(* CODESYS project SNDLTN_HTTP.library
   Author: S. Verbeek
   Title: SNDLTN_HTTP
   Version: 1.2.200929
   Description: Library created to ease the use of the CoDeSys HTTP example.
   Company: Sandolution

Project tree, tasks and I/O mapping:
  libraries: CAA Net Base Services, * (CAA Technical Workgroup); CAA Behaviour Model, * (CAA Technical Workgroup); StringUtils, * (System); CAA Types, 3.0.0.1 (CAA Technical Workgroup)
  Constants/
    global variables HTTP_UTF8
    global variables HTTP_Properties
    global variables HTTP_Constants
  Enums/
    data type HTTP_eRequestType
    data type HTTP_eContentType
    data type HTTP_eError
    data type HTTP_eState_int
  Function Blocks/
    function block HTTP_Client [ST]: prvStart, StringToURL, prvCyclicAction, prvResetOutputs, CreateRequest, Close, prvAbort, ParseResult
  Functions/
    function HTTP_UTF8toUTF16_3S [ST]
    function HTTP_UTF16toUTF8_3S [ST]
    function HTTP_Concat_3S [ST]
    function HTTP_IsLegalUTF8_3S [ST]
  Structs/
    data type HTTP_scResponse
    data type HTTP_scURL_int
  Variables/
  program ChangeLog [ST]
*)

// Enums/HTTP_eRequestType
{attribute 'qualified_only'}
TYPE HTTP_eRequestType :
(
	GET := 0,
	POST, 		//(Requires pwsPostValue) 
	DELETE, 
	PUT,		//(Requires pwsPostValue) 
	HEAD
);
END_TYPE

// Enums/HTTP_eContentType
{attribute 'qualified_only'}
TYPE HTTP_eContentType :
(
	FORM := 0,		//HTTP FORM DATA
	JSON			//JSON/XML format
);
END_TYPE

// Enums/HTTP_eError
{attribute 'qualified_only'}
{attribute 'to_string'}
TYPE HTTP_eError :
(
	NoError 					:= 0, 		// No error
	
	//1000-1999 : HTTP ERRORS
	TCPInitError				:= 1001, 	// Unable to initialize the TCP socket
	TCPReadError				:= 1002, 	// Error while reading response
	TCPWriteError				:= 1003, 	// Error while sending the request
	MissingPostValue			:= 1004, 	// Current request type needs a post value
	ParsingError				:= 1005, 	// Error while parsing the response
	
	//NBS errors (ported from 6001-6099)
	NBS_TimeOut 				:= 1100,	//Time limit exceeded
	NBS_InvalidAddress			:= 1101,	//Address invalid
	NBS_InvalidHandle			:= 1102,	//Handle invalid
	NBS_InvalidPointer			:= 1103,	//Data pointer invalid
	NBS_InvalidSize				:= 1104,	//Data size invalid
	NBS_ReceiveUDP				:= 1105,	//Error receiving data via UDP
	NBS_SendUDP					:= 1106,	//Error sending data via UDP
	NBS_SentIncompleteUDP		:= 1107,	//Not all data is sent.
	NBS_OpenUDP					:= 1108,	//Couldn't open UDP connection
	NBS_CloseUDP				:= 1109,	//Couldn't close UDP connection
	NBS_SendTCP					:= 1110,	//Error sending data via TCP
	NBS_ReceiveTCP				:= 1111,	//Error receiving data via TCP
	NBS_OpenTCP					:= 1112,	//Couldn't open TCP connection
	NBS_ConnectTCP				:= 1113,	//Couldn't connect TCP connection
	NBS_CloseTCP				:= 1114,	//Couldn't close TCP connection
	NBS_ServerTCP				:= 1115,	//Server error TCP
	NBS_WrongParameter			:= 1116,	//Wrong parameters entered
	NBS_Unknown					:= 1117		//Not specified
);
END_TYPE

// Enums/HTTP_eState_int
{attribute 'qualified_only'}
{attribute 'conditionalshow'}
TYPE HTTP_eState_int :
(
	Start 	:= 0,
	Init,
	Request,
	Response,
	Error,
	Idle
);
END_TYPE

// Structs/HTTP_scResponse
TYPE HTTP_scResponse :
STRUCT
	iStatus				: INT; // http status
	wsHeader			: WSTRING(HTTP_Properties.uiHTTPMaxHeaderSize); 	//http header as WSTRING
	wsContent			: WSTRING(HTTP_Properties.uiHTTPMaxResponseSize); //The result of the request as WSTRING
	sHeader				: STRING(HTTP_Properties.uiHTTPMaxHeaderSize); 	//http header as STRING
	sContent			: STRING(HTTP_Properties.uiHTTPMaxResponseSize); 	//The result of the request as STRING
	diContentLength		: DINT; // Length of wsContent
END_STRUCT
END_TYPE

// Structs/HTTP_scURL_int
{attribute 'hide'}
TYPE HTTP_scURL_int :
STRUCT
	wsProtocol	: WSTRING(5); 	// Protocol e.g. http, NOTE: ONLY HTTP IS SUPPORTED! 
	wsDomain	: WSTRING(255); 	// The domain e.g. 'twitter.api.com'
	uiPort		: UINT;			// Port of the server
	wsPath		: WSTRING(255);	// The path e.g. '/1.1/statuses/update.json'
END_STRUCT
END_TYPE

// Constants/HTTP_UTF8
{attribute 'qualified_only'}
{attribute 'conditionalshow'}
VAR_GLOBAL CONSTANT
	trailingBytesForUTF8 	: ARRAY[0..255] OF BYTE := [
							0,0,0,0,0,0,0,0,0,0,0,0,0,0,0,0, 0,0,0,0,0,0,0,0,0,0,0,0,0,0,0,0,
							0,0,0,0,0,0,0,0,0,0,0,0,0,0,0,0, 0,0,0,0,0,0,0,0,0,0,0,0,0,0,0,0,
							0,0,0,0,0,0,0,0,0,0,0,0,0,0,0,0, 0,0,0,0,0,0,0,0,0,0,0,0,0,0,0,0,
							0,0,0,0,0,0,0,0,0,0,0,0,0,0,0,0, 0,0,0,0,0,0,0,0,0,0,0,0,0,0,0,0,
							0,0,0,0,0,0,0,0,0,0,0,0,0,0,0,0, 0,0,0,0,0,0,0,0,0,0,0,0,0,0,0,0,
							0,0,0,0,0,0,0,0,0,0,0,0,0,0,0,0, 0,0,0,0,0,0,0,0,0,0,0,0,0,0,0,0,
							1,1,1,1,1,1,1,1,1,1,1,1,1,1,1,1, 1,1,1,1,1,1,1,1,1,1,1,1,1,1,1,1,
							2,2,2,2,2,2,2,2,2,2,2,2,2,2,2,2, 3,3,3,3,3,3,3,3,4,4,4,4,5,5,5,5
							];
							
	firstByteMark 			: ARRAY[0..6] OF BYTE := [ 16#00, 16#00, 16#C0, 16#E0, 16#F0, 16#F8, 16#FC ];
	
	offsetsFromUTF8			: ARRAY[0..5] OF DWORD := [16#00000000, 16#00003080, 16#000E2080, 16#03C82080, 16#FA082080, 16#82082080];
	
	halfShift				: INT := 10; (* used FOR shifting BY 10 bits *)

	halfBase 				: DWORD := 16#0010000;
	halfMask 				: DWORD := 16#3FF;
	
	UNI_REPLACEMENT_CHAR 	: DWORD := 16#0000FFFD;
	
	UNI_MAX_BMP 			: DWORD := 16#0000FFFF;
	UNI_MAX_UTF16			: DWORD := 16#0010FFFF;
	
	byteMask 				: DWORD := 16#BF;
	byteMark				: DWORD := 16#80;
	UNI_SUR_HIGH_START 		: DWORD := 16#D800;
 	UNI_SUR_HIGH_END 		: DWORD := 16#DBFF;
 	UNI_SUR_LOW_START 		: DWORD := 16#DC00;
 	UNI_SUR_LOW_END 		: DWORD := 16#DFFF;
	
	ERR_OK 					: UDINT := 16#0000;	(* The operation succeeded *)
	ERR_SOURCE_EXHAUSTED 	: UDINT := 16#40A0; (* Used for UTF8 helper *)
	ERR_TARGET_EXHAUSTED 	: UDINT := 16#40A1; (* Used for UTF8 helper *)
	ERR_SOURCE_ILLEGAL 		: UDINT := 16#40A2; (* Used for UTF8 helper *)
	
END_VAR

// Constants/HTTP_Properties
{attribute 'qualified_only'}
{attribute 'analysis' := '-33'}
VAR_GLOBAL CONSTANT
	uiHTTPMaxURLSize			: UINT := 512;
	uiHTTPMaxResponseSize		: UINT := 16384;
	uiHTTPMaxRequestSize		: UINT := 8192;
	uiHTTPMaxHeaderSize			: UINT := 4096;
END_VAR
{attribute 'analysis' := '+33'}

// Constants/HTTP_Constants
{attribute 'qualified_only'}
{attribute 'conditionalshow'}
VAR_GLOBAL
	wsBLANK 					: WSTRING(1) := " ";
	wsDoubleDash				: WSTRING(1) := ":";
	wsLF						: WSTRING(2) :=	"$R$N";
	wsDoubleLF					: WSTRING(4) :=	"$R$N$R$N";
	wsChunked					: WSTRING(26) := "Transfer-Encoding: chunked";
	wsHex						: WSTRING(3) :=	"16#";
END_VAR

// Function Blocks/HTTP_Client
// Functionblock to send http GET and POST requests.
{attribute 'conditionalshow_all_locals'}
FUNCTION_BLOCK HTTP_Client EXTENDS CBM.ETrigTo
VAR_INPUT
	sURL					:STRING(HTTP_Properties.uiHTTPMaxURLSize); // URL of the web server
	eRequestType			:HTTP_eRequestType := HTTP_eRequestType.GET;	//Type of the request
	eContentType			:HTTP_eContentType := HTTP_eContentType.JSON; 	//Content-Type of the request
	pwsAdditionalHeader		:POINTER TO WSTRING; // Additional HTTP header
	pwsPostValue			:POINTER TO WSTRING; // Post parameter
END_VAR                      
VAR_OUTPUT                   
	xResponseValid			:BOOL;              
	eErrorID				:HTTP_eError; // Current error state
	scResponse				:HTTP_scResponse; // The result of the request
END_VAR                       
VAR                           
	// TCP Connection         
	_tcp_client 			:NBS.TCP_Client;
	_tcp_read 				:NBS.TCP_Read;
	_tcp_write 				:NBS.TCP_Write;
	_IPAddr 				:NBS.IP_ADDR;	
	_wsRequest 				:WSTRING(HTTP_Properties.uiHTTPMaxRequestSize);
	_abRequest 				:ARRAY[0..HTTP_Properties.uiHTTPMaxRequestSize] OF BYTE;
	_sContent				:STRING(HTTP_Properties.uiHTTPMaxResponseSize); 
	_pbContent				:POINTER TO BYTE;
	_wsContent				:WSTRING(HTTP_Properties.uiHTTPMaxResponseSize);
	_url					:HTTP_scURL_int;
	// Helpers	             
	_eState 				:HTTP_eState_int;	

	diContentLength			:DINT;
	diStringLength			:DINT;
END_VAR

//Call CoDeSys functions
SUPER^();

//Write error outputs
IF _tcp_client.xError THEN
	eErrorID := _tcp_client.eError - 4900;	//NBS starts at 6000 > SNDLTN_MQTT at 1000 > -5000
ELSIF _tcp_read.xError THEN
	eErrorID := _tcp_read.eError - 4900;		//NBS starts at 6000 > SNDLTN_MQTT at 1000 > -5000
ELSIF _tcp_write.xError THEN
	eErrorID := _tcp_write.eError - 4900;		//NBS starts at 6000 > SNDLTN_MQTT at 1000 > -5000
ELSIF iError <> 0 THEN
	eErrorID := iError;
ELSE
	eErrorID := HTTP_eError.NoError;
END_IF
//Overrule CoDeSys implementation
xError := eErrorID <> HTTP_eError.NoError;

//Response within range
xResponseValid := scResponse.diContentLength >= (diContentLength-16) AND scResponse.diContentLength <= (diContentLength+16);

{attribute 'conditionalshow'}
METHOD prvStart : BOOL
VAR_INPUT
END_VAR
VAR
END_VAR
END_METHOD

{attribute 'conditionalshow'}
// Converts a string to an url.
METHOD StringToURL : HTTP_eError
VAR_INPUT
	wsUrl			:WSTRING(1024);	// The url as string
END_VAR         	 
VAR_IN_OUT      	 
	url				:HTTP_scURL_int; // The URL struct
END_VAR         	 
VAR             	 
	wsTemp			:WSTRING(1024);
	wsPort			:WSTRING(6);
	i				:INT;
END_VAR         	
VAR CONSTANT    	
	wsDel			:WSTRING(3) := "://";
	wsPortDel		:WSTRING(1) := ":";
	wsPathStart		:WSTRING(1) := "/";
END_VAR
// Find '://'
i := Stu.StrFindW(pst1 := ADR(wsUrl), pst2 := ADR(wsDel), uiSearchStart := 1);
IF i > 0 THEN
	Stu.StrMidW(pwst := ADR(wsUrl),
				uiInputBufferSize := SIZEOF(wsUrl),
				iLength := DINT_TO_INT(Stu.StrLenW(ADR(wsUrl))) - i - DINT_TO_INT(Stu.StrLenW(ADR(wsDel))) + 1,
				iPosition := i +  DINT_TO_INT(Stu.StrLenW(ADR(wsDel))),
				pwstResult := ADR(wsTemp),
				uiResultBufferSize := SIZEOF(wsTemp));
	// Set protocol			
	Stu.StrMidW(pwst := ADR(wsUrl),
				uiInputBufferSize := SIZEOF(wsUrl),
				iLength := i - 1,
				iPosition := 1,
				pwstResult := ADR(url.wsProtocol),
				uiResultBufferSize := SIZEOF(url.wsProtocol));
ELSE
	url.wsProtocol := "http";
	wsTemp := wsUrl;
END_IF

// Find path start '/'
i := Stu.StrFindW(pst1 := ADR(wsTemp), pst2 := ADR(wsPathStart), uiSearchStart := 1);
IF i > 0 THEN
	// set path
	Stu.StrMidW(pwst := ADR(wsTemp),
				uiInputBufferSize := SIZEOF(wsTemp),
				iLength := DINT_TO_INT(Stu.StrLenW(ADR(wsTemp))) - i + DINT_TO_INT(Stu.StrLenW(ADR(wsPathStart))),
				iPosition := i + DINT_TO_INT(Stu.StrLenW(ADR(wsPathStart))) - 1,
				pwstResult := ADR(url.wsPath),
				uiResultBufferSize := SIZEOF(url.wsPath));	
				
	Stu.StrMidW(pwst := ADR(wsTemp),
				uiInputBufferSize := SIZEOF(wsTemp),
				iLength := i - 1,
				iPosition := 1,
				pwstResult := ADR(wsTemp),
				uiResultBufferSize := SIZEOF(wsTemp));			
ELSE
	url.wsPath := "";
END_IF


i := Stu.StrFindW(pst1 := ADR(wsTemp), pst2 := ADR(wsPortDel), uiSearchStart := 1);
IF i > 0 THEN
	// set domain
	Stu.StrMidW(pwst := ADR(wsTemp),
				uiInputBufferSize := SIZEOF(wsTemp),
				iLength := i - 1,
				iPosition := 1,
				pwstResult := ADR(url.wsDomain),
				uiResultBufferSize := SIZEOF(url.wsDomain));	
	// set port
	Stu.StrMidW(pwst := ADR(wsTemp),
				uiInputBufferSize := SIZEOF(wsTemp),
				iLength := DINT_TO_INT(Stu.StrLenW(ADR(wsTemp)) - i - Stu.StrLenW(ADR(wsPortDel))) + 1,
				iPosition := i + DINT_TO_INT(Stu.StrLenW(ADR(wsPortDel))),
				pwstResult := ADR(wsPort),
				uiResultBufferSize := SIZEOF(wsPort));
	url.uiPort := WSTRING_TO_UINT(wsPort);				
ELSE
	url.wsDomain := wsTemp;
	url.uiPort := 80;
END_IF

IF url.wsPath = "" THEN
	url.wsPath := "/";
END_IF
END_METHOD

{attribute 'conditionalshow'}
METHOD prvCyclicAction : BOOL
VAR_INPUT
END_VAR
VAR
	uxiBytesRead		:__UXINT;
END_VAR

IF xExecute = TRUE AND _eState = HTTP_eState_int.Idle THEN
	_eState := HTTP_eState_int.Start;
END_IF

CASE _eState OF
	
HTTP_eState_int.Idle: // Idle

HTTP_eState_int.Start: // stopped
	// Parse url 
	_sContent := '';
	_pbContent := ADR(_sContent);
	_wsContent := "";
	scResponse.wsContent := "";
	scResponse.wsHeader := "";
	scResponse.diContentLength := 0;
	scResponse.iStatus := 0;
	StringToURL(wsUrl := STRING_TO_WSTRING(sUrl), url := _url);
	_IPAddr.sAddr := WSTRING_TO_STRING(_url.wsDomain);
	_tcp_client(xEnable := FALSE);
	_tcp_read(xEnable := FALSE);
	_tcp_write(xExecute := FALSE);
	_eState := HTTP_eState_int.Init;
	IF (eRequestType = HTTP_eRequestType.POST OR eRequestType = HTTP_eRequestType.PUT) AND (pwsPostValue = 0 OR Stu.StrLenW(pstData := pwsPostValue) = 0) THEN
		iError := HTTP_eError.MissingPostValue;
		_eState := HTTP_eState_int.Error;
	END_IF
	
HTTP_eState_int.Init:	// init client
	_tcp_client(xEnable := TRUE, ipAddr := _IPAddr, uiPort := _url.uiPort);
	IF _tcp_client.xBusy AND _tcp_client.hConnection <> CAA.gc_hINVALID THEN
		_eState := HTTP_eState_int.Request;
	ELSIF _tcp_client.xError THEN
		iError := HTTP_eError.TCPInitError;
		_eState := HTTP_eState_int.Error;
	END_IF
	
HTTP_eState_int.Request:		// send message	
	CreateRequest(url := _url, pwsAdditionalHeader := pwsAdditionalHeader, pwsPostValue := pwsPostValue, wsOut := _wsRequest);
	HTTP_UTF16toUTF8_3S(pwSourceStart := ADR(_wsRequest), pbyTargetStart := ADR(_abRequest), dwTargetBufferSize := SIZEOF(_abRequest), xStrictConversion := FALSE);
	_tcp_write(xExecute := _tcp_client.xActive, hConnection := _tcp_client.hConnection, szSize := DINT_TO_UDINT(Stu.StrLenA(ADR(_abRequest))), pData := ADR(_abRequest));
	IF _tcp_write.xDone THEN		// message sent, go back to idle mode
		_tcp_write(xExecute := FALSE);			
		_eState := HTTP_eState_int.Response;
	ELSIF _tcp_write.xError THEN
		iError := HTTP_eError.TCPWriteError;
		_eState := HTTP_eState_int.Error;
	END_IF
	
HTTP_eState_int.Response:	// idle mode - wait for incomming message
	_tcp_read(xEnable := _tcp_client.xActive, hConnection := _tcp_client.hConnection, szSize := SIZEOF(_sContent), pData := ADR(_sContent), szCount => uxiBytesRead);
	IF _tcp_read.xReady THEN		
		_pbContent[uxiBytesRead] := 0;
		_tcp_read(xEnable := FALSE);		
		_eState := HTTP_eState_int.Idle;
		Close();
		HTTP_UTF8toUTF16_3S(pbySourceStart := ADR(_sContent), pbyTargetStart := ADR(_wsContent), dwTargetBufferSize := SIZEOF(_wsContent), xStrictConversion := FALSE);
		ParseResult(wsContent := _wsContent, scResponse := scResponse);
		xDone := TRUE;
	ELSIF _tcp_read.xError THEN		
		iError := HTTP_eError.TCPReadError;
		_eState := HTTP_eState_int.Error;		
		xError := TRUE;	
	END_IF		

HTTP_eState_int.Error:
	_sContent := '';
	_wsContent := "";
	Close();
	_eState := HTTP_eState_int.Idle;
	
END_CASE
END_METHOD

{attribute 'conditionalshow'}
METHOD prvResetOutputs : BOOL
VAR_INPUT
END_VAR
VAR
END_VAR
SUPER^.prvResetOutputs();
END_METHOD

// Builds a http request
{attribute 'conditionalshow'}
METHOD CreateRequest
VAR_INPUT
	url						:HTTP_scURL_int; // The URL of the webserver
	pwsAdditionalHeader		:POINTER TO WSTRING; // Additional HTTP header	
	pwsPostValue			:POINTER TO WSTRING; // Post parameter
END_VAR                      
VAR_IN_OUT                   
	wsOut					:WSTRING(HTTP_Properties.uiHTTPMaxRequestSize);
END_VAR                      
VAR                          
	wsType					:WSTRING(6); // Type of the request: GET or POST
	wsContentLength			:WSTRING(5);
	wsHTTP_HEADER			:WSTRING(100) 	:= "Connection: close$000D$000AContent-Type: application/x-www-form-urlencoded";
END_VAR
VAR CONSTANT
	wsBlank					:WSTRING(1) 	:= " ";
	wsLF					:WSTRING(2) 	:= "$000D$000A";
	wsHTTPVersion			:WSTRING(12) 	:= " HTTP/1.1";
	wsHTTPContetntLength	:WSTRING(17) 	:= "Content-Length: ";
	wsHTTPHost 				:WSTRING(9) 	:= "Host: ";
END_VAR
IF eRequestType = HTTP_eRequestType.GET THEN
	wsType := "GET";
ELSIF eRequestType = HTTP_eRequestType.DELETE THEN
	wsType := "DELETE";
ELSIF eRequestType = HTTP_eRequestType.HEAD THEN
	wsType := "HEAD";
ELSIF eRequestType = HTTP_eRequestType.PUT THEN
	wsType := "PUT";
ELSIF eRequestType = HTTP_eRequestType.POST THEN
	wsType := "POST";
ELSE
	wsType := "";
END_IF

IF eContentType = HTTP_eContentType.JSON THEN
	wsHTTP_HEADER := "Connection: close$000D$000AContent-Type: application/json";
ELSE
	wsHTTP_HEADER := "Connection: close$000D$000AContent-Type: application/x-www-form-urlencoded";
END_IF

// POST or GET
wsOut := "";
HTTP_Concat_3S(ADR(wsType), ADR(wsOut), SIZEOF(wsOut));
HTTP_Concat_3S(ADR(wsBlank), ADR(wsOut), SIZEOF(wsOut));
HTTP_Concat_3S(ADR(url.wsPath), ADR(wsOut), SIZEOF(wsOut));
HTTP_Concat_3S(ADR(wsHTTPVersion), ADR(wsOut), SIZEOF(wsOut));
HTTP_Concat_3S(ADR(wsLF), ADR(wsOut), SIZEOF(wsOut));

// HTTP Header
Stu.StrConcatW(ADR(wsHTTP_HEADER), ADR(wsOut), DINT_TO_INT(SIZEOF(wsOut)));
Stu.StrConcatW(ADR(wsLF), ADR(wsOut), DINT_TO_INT(SIZEOF(wsOut)));
IF NOT Stu.StrIsNullOrEmptyA(pwsAdditionalHeader) THEN
	Stu.StrConcatW(pwsAdditionalHeader, ADR(wsOut), DINT_TO_INT(SIZEOF(wsOut)));
	Stu.StrConcatW(ADR(wsLF), ADR(wsOut), DINT_TO_INT(SIZEOF(wsOut)));
END_IF

// Host
HTTP_Concat_3S(ADR(wsHTTPHost), ADR(wsOut), SIZEOF(wsOut));
HTTP_Concat_3S(ADR(url.wsDomain), ADR(wsOut), SIZEOF(wsOut));
HTTP_Concat_3S(ADR(wsLF), ADR(wsOut), SIZEOF(wsOut));

IF eRequestType = HTTP_eRequestType.POST OR eRequestType = HTTP_eRequestType.PUT THEN
	HTTP_Concat_3S(ADR(wsHTTPContetntLength), ADR(wsOut), SIZEOF(wsOut));
	wsContentLength := DINT_TO_WSTRING(Stu.StrLenW(pwsPostValue));
	HTTP_Concat_3S(ADR(wsContentLength), ADR(wsOut), SIZEOF(wsOut));
END_IF
HTTP_Concat_3S(ADR(wsLF), ADR(wsOut), SIZEOF(wsOut));
HTTP_Concat_3S(ADR(wsLF), ADR(wsOut), SIZEOF(wsOut));

// Post content
IF eRequestType = HTTP_eRequestType.POST OR eRequestType = HTTP_eRequestType.PUT THEN
	HTTP_Concat_3S(pwsPostValue, ADR(wsOut), SIZEOF(wsOut));
END_IF
END_METHOD

{attribute 'conditionalshow'}
METHOD Close
VAR_INPUT
END_VAR
_tcp_write(xExecute := FALSE);	
_tcp_read(xEnable := FALSE);	
_tcp_client(xEnable := FALSE);
END_METHOD

{attribute 'conditionalshow'}
METHOD prvAbort : BOOL
VAR_INPUT
END_VAR
VAR
END_VAR
Close();
_eState := HTTP_eState_int.Idle;
xAbortInProgress := FALSE;
END_METHOD

{attribute 'conditionalshow'}
METHOD ParseResult : HTTP_eError
VAR_IN_OUT
	wsContent 				:WSTRING(HTTP_Properties.uiHTTPMaxResponseSize);
	scResponse 				:HTTP_scResponse;
END_VAR                 	
VAR                     	
	diTemp1 				:DINT;
	diTemp2 				:DINT;
	diContentStartPos 		:DINT;
	wsStatus 				:WSTRING(4);
	wsContentLength 		:WSTRING(20);
	wsContentLengthHex 		:WSTRING(20);
	xIsChunked				:BOOL;
	wsContentLenghtHeader	:WSTRING(HTTP_Properties.uiHTTPMaxHeaderSize);
END_VAR
//Reset output
scResponse.diContentLength := 0;
scResponse.wsHeader := "";
scResponse.wsContent := "";
scResponse.sHeader := '';
scResponse.sContent := '';

// Find HTTP status
diTemp1 := StrFindW(pst1 := ADR(wsContent), pst2 := ADR(HTTP_Constants.wsBLANK), uiSearchStart := 0);
diTemp2 := StrFindW(pst1 := ADR(wsContent), pst2 := ADR(HTTP_Constants.wsBLANK), uiSearchStart := DINT_TO_UINT(diTemp1 + 1));
IF diTemp1 < 1 OR diTemp2 < 1 THEN
	ParseResult := HTTP_eError.ParsingError;
	RETURN;
END_IF
StrMidW(pwst := ADR(wsContent), 
		uiInputBufferSize := SIZEOF(wsContent), 
		iLength := DINT_TO_INT(diTemp2 - diTemp1), 
		iPosition := DINT_TO_INT(diTemp1), 
		pwstResult := ADR(wsStatus), 
		uiResultBufferSize := SIZEOF(wsStatus));
scResponse.iStatus := WSTRING_TO_INT(wsStatus);

// Find header
diTemp1 := StrFindW(pst1 := ADR(wsContent), pst2 := ADR(HTTP_Constants.wsLF), uiSearchStart := DINT_TO_UINT(diTemp2 + 1));
diTemp2 := StrFindW(pst1 := ADR(wsContent), pst2 := ADR(HTTP_Constants.wsDoubleLF), uiSearchStart := DINT_TO_UINT(diTemp1 + 1));
IF diTemp1 < 1 OR diTemp2 < 1 THEN
	ParseResult := HTTP_eError.ParsingError;
	RETURN;
END_IF
StrMidW(pwst := ADR(wsContent), 
		uiInputBufferSize := SIZEOF(wsContent), 
		iLength := DINT_TO_INT(diTemp2 - diTemp1) - 2, 
		iPosition := DINT_TO_INT(diTemp1) + 2, 
		pwstResult := ADR(scResponse.wsHeader), 
		uiResultBufferSize := SIZEOF(scResponse.wsHeader));

diContentStartPos := diTemp2 + 4;

xIsChunked := StrFindW(pst1 := ADR(scResponse.wsHeader), pst2 := ADR(HTTP_Constants.wsChunked), uiSearchStart := 0) > 0;
IF xIsChunked THEN
	// Convert chunked data
	diTemp1 := diContentStartPos;
	// Get data length
	diTemp2 := StrFindW(pst1 := ADR(wsContent), pst2 := ADR(HTTP_Constants.wsLF), uiSearchStart := DINT_TO_UINT(diTemp1));
	IF diTemp2 < 1 THEN
		ParseResult := HTTP_eError.ParsingError;
		RETURN;
	END_IF
	StrMidW(pwst := ADR(wsContent), 
			uiInputBufferSize := SIZEOF(wsContent), 
			iLength := DINT_TO_INT(diTemp2 - diTemp1), 
			iPosition := DINT_TO_INT(diTemp1), 
			pwstResult := ADR(wsContentLength), 
			uiResultBufferSize := SIZEOF(wsContentLength));
	wsContentLengthHex := HTTP_Constants.wsHex;
	StrConcatW(pstFrom := ADR(wsContentLength), pstTo := ADR(wsContentLengthHex), iBufferSize := TO_INT(SIZEOF(wsContentLengthHex)));
	scResponse.diContentLength := WSTRING_TO_DINT(wsContentLengthHex);
	// Copy content
	StrMidW(pwst := ADR(wsContent), 
			uiInputBufferSize := SIZEOF(wsContent), 
			iLength := DINT_TO_INT(scResponse.diContentLength), 
			iPosition := DINT_TO_INT(diTemp2 + 2), 
			pwstResult := ADR(scResponse.wsContent), 
			uiResultBufferSize := SIZEOF(scResponse.wsContent));
ELSE	
	// Find content
	diTemp2 := StrLenW(pstData := ADR(wsContent));
	IF diTemp2 < 0 THEN
		ParseResult := HTTP_eError.ParsingError;
		RETURN;
	END_IF
	StrMidW(pwst := ADR(wsContent), 
			uiInputBufferSize := SIZEOF(wsContent), 
			iLength := DINT_TO_INT(diTemp2 - diContentStartPos), 
			iPosition := DINT_TO_INT(diContentStartPos), 
			pwstResult := ADR(scResponse.wsContent), 
			uiResultBufferSize := SIZEOF(scResponse.wsContent));
	scResponse.diContentLength := diTemp2 - diContentStartPos;
END_IF

// Copy WSTRING to STRING values
HTTP_UTF16toUTF8_3S(pwSourceStart := ADR(scResponse.wsHeader), pbyTargetStart := ADR(scResponse.sHeader), dwTargetBufferSize := SIZEOF(scResponse.sHeader), xStrictConversion := FALSE);
HTTP_UTF16toUTF8_3S(pwSourceStart := ADR(scResponse.wsContent), pbyTargetStart := ADR(scResponse.sContent), dwTargetBufferSize := SIZEOF(scResponse.sContent), xStrictConversion := FALSE);

//Get string length
diStringLength := StrLenW(pstData := ADR(scResponse.sContent));

//Get content length
diTemp1 := StrFindW(pst1 := ADR(scResponse.wsHeader), pst2 := ADR(HTTP_Constants.wsLF), uiSearchStart := 1);	//$R$N
diTemp2 := StrFindW(pst1 := ADR(scResponse.wsHeader), pst2 := ADR(HTTP_Constants.wsDoubleDash), uiSearchStart := 1);	//:
StrMidW(pwst := ADR(scResponse.wsHeader), 
		uiInputBufferSize := SIZEOF(scResponse.wsHeader), 
		iLength := TO_INT(diTemp1-diTemp2)-2, 
		iPosition := TO_INT(diTemp2+2), 
		pwstResult := ADR(wsContentLenghtHeader), 
		uiResultBufferSize := SIZEOF(wsContentLenghtHeader));
		
diContentLength := TO_DINT(wsContentLenghtHeader);
END_METHOD

END_FUNCTION_BLOCK

// Functions/HTTP_UTF16toUTF8_3S
{attribute 'conditionalshow'}
// Converts a WSTRING to STRING
FUNCTION HTTP_UTF16toUTF8_3S : UDINT
VAR_INPUT
 	pwSourceStart 		: POINTER TO WORD;	// Pointer to WSTRING
	pbyTargetStart 		: POINTER TO BYTE;	// Pointer to STRING
	dwTargetBufferSize 	: DWORD;		// Size of STRING
	xStrictConversion 	: BOOL;
END_VAR
VAR
	pwSource 			: POINTER TO WORD;
	pwSourceEnd 		: POINTER TO WORD;
	pwSourceOld 		: POINTER TO WORD;
	pbyTarget 			: POINTER TO BYTE;
	pbyTargetEnd 		: POINTER TO BYTE;
	dwSource_1 			: DWORD;
	dwSource_2 			: DWORD;
	wBytesToWrite 		: WORD := 0;
	wBytesToWriteSave 	: WORD := 0;
END_VAR

HTTP_UTF16toUTF8_3S := HTTP_UTF8.ERR_OK;
pwSource := pwSourceStart;
pbyTarget := pbyTargetStart;
pwSourceEnd := pwSource + TO_WORD(StrLenW(pwSource))*2 + 1; // Add the terminating 0
pbyTargetEnd := pbyTarget + dwTargetBufferSize;
WHILE pwSource < pwSourceEnd DO
	wBytesToWrite := 0;
    pwSourceOld := pwSource; // In CASE we have TO back up because OF target overflow.
    dwSource_1 := WORD_TO_DWORD(pwSource^);
	pwSource := pwSource + 2;
    (* If we have a surrogate pair, convert to UTF32 first. *)
    IF (dwSource_1 >= HTTP_UTF8.UNI_SUR_HIGH_START AND dwSource_1 <= HTTP_UTF8.UNI_SUR_HIGH_END) THEN
        (* If the 16 bits following the high surrogate are in the source buffer... *)
        IF (pwSource < pwSourceEnd) THEN
        	dwSource_2 := WORD_TO_DWORD(pwSource^);
        	(* If it's a low surrogate, convert to UTF32. *)
			IF (dwSource_2 >= HTTP_UTF8.UNI_SUR_LOW_START AND dwSource_2 <= HTTP_UTF8.UNI_SUR_LOW_END) THEN
				dwSource_1 := SHL(dwSource_1 - HTTP_UTF8.UNI_SUR_HIGH_START, HTTP_UTF8.halfShift) + (dwSource_2 - HTTP_UTF8.UNI_SUR_LOW_START) + HTTP_UTF8.halfBase;
				pwSource := pwSource + 2;
			ELSIF (xStrictConversion) THEN
				(* it's an unpaired high surrogate *)
				pwSource := pwSource - 2; // return to the illegal value itself 
				HTTP_UTF16toUTF8_3S := HTTP_UTF8.ERR_SOURCE_ILLEGAL;
				EXIT;
			END_IF
		ELSE 
		 	(* We don't have the 16 bits following the high surrogate. *)
			pwSource := pwSource - 2; // return to the high surrogate
			HTTP_UTF16toUTF8_3S := HTTP_UTF8.ERR_SOURCE_EXHAUSTED;
			EXIT;
		END_IF
	ELSIF (xStrictConversion) THEN
        (* UTF-16 surrogate values are illegal in UTF-32 *)
        IF (dwSource_1 >= HTTP_UTF8.UNI_SUR_LOW_START AND dwSource_1 <= HTTP_UTF8.UNI_SUR_LOW_END) THEN
        	pwSource := pwSource - 2; // RETURN TO the illegal value itself
        	HTTP_UTF16toUTF8_3S := HTTP_UTF8.ERR_SOURCE_ILLEGAL;
        	EXIT;
        END_IF
    END_IF
    (* Figure out how many bytes the result will require *)
    IF (dwSource_1 < 16#80) THEN      
		wBytesToWrite := 1;
    ELSIF (dwSource_1 < 16#800) THEN     
		wBytesToWrite := 2;
    ELSIF (dwSource_1 < 16#10000) THEN   
		wBytesToWrite := 3;
    ELSIF (dwSource_1 < 16#110000) THEN  
		wBytesToWrite := 4;
    ELSE       
		wBytesToWrite := 3;
        dwSource_1 := HTTP_UTF8.UNI_REPLACEMENT_CHAR;
    END_IF

    pbyTarget := pbyTarget + wBytesToWrite;
    IF (pbyTarget > pbyTargetEnd) THEN
        pwSource := pwSourceOld; // Back up source pointer! 
        pbyTarget := pbyTarget - wBytesToWrite; 
		HTTP_UTF16toUTF8_3S := HTTP_UTF8.ERR_TARGET_EXHAUSTED; 
		EXIT;
   	END_IF
	wBytesToWriteSave := wBytesToWrite;
    IF wBytesToWrite = 4 THEN
		pbyTarget := pbyTarget - 1;
		pbyTarget^ := DWORD_TO_BYTE((dwSource_1 OR HTTP_UTF8.byteMark) AND HTTP_UTF8.byteMask); 
		dwSource_1 := SHR(dwSource_1, 6);
		wBytesToWrite := 3;
	END_IF
	IF wBytesToWrite = 3 THEN
		pbyTarget := pbyTarget - 1;
		pbyTarget^ := DWORD_TO_BYTE((dwSource_1 OR HTTP_UTF8.byteMark) AND HTTP_UTF8.byteMask); 
		dwSource_1 := SHR(dwSource_1, 6);
		wBytesToWrite := 2;
	END_IF
	IF wBytesToWrite = 2 THEN
		pbyTarget := pbyTarget - 1;
		pbyTarget^ := DWORD_TO_BYTE((dwSource_1 OR HTTP_UTF8.byteMark) AND HTTP_UTF8.byteMask); 
		dwSource_1 := SHR(dwSource_1, 6);
		wBytesToWrite := 1;
	END_IF
	IF wBytesToWrite = 1 THEN
		pbyTarget := pbyTarget - 1;
		pbyTarget^ := DWORD_TO_BYTE(dwSource_1 OR HTTP_UTF8.firstByteMark[wBytesToWriteSave]);
	END_IF
    pbyTarget := pbyTarget + wBytesToWriteSave;
END_WHILE

END_FUNCTION

// Functions/HTTP_UTF8toUTF16_3S
{attribute 'conditionalshow'}
// Converts a STRING to WSTRING.
FUNCTION HTTP_UTF8toUTF16_3S : UDINT
VAR_INPUT
 	pbySourceStart 			: POINTER TO BYTE; 	// Pointer to STRING
	pbyTargetStart 			: POINTER TO WORD;	// Pointer to WSTRING
	dwTargetBufferSize 		: DWORD;		// Size of the WSTRING
	xStrictConversion 		: BOOL;
END_VAR                 	
VAR                     	
	pbySource 				: POINTER TO BYTE;
	pbySourceEnd 			: POINTER TO BYTE;
	pwTarget 				: POINTER TO WORD;
	pwTargetEnd 			: POINTER TO WORD;
	dwSource 				: DWORD;
	wExtraBytesToRead 		: WORD;
	wExtraBytesToReadSave	: WORD;
END_VAR

HTTP_UTF8toUTF16_3S := HTTP_UTF8.ERR_OK;
pbySource := pbySourceStart;
pwTarget := pbyTargetStart;
pbySourceEnd := pbySource + TO_DWORD(StrLenA(pbySource)) + 1; // Add the terminating 0 
pwTargetEnd := pwTarget + dwTargetBufferSize;
WHILE (pbySource < pbySourceEnd) DO
	dwSource := 0;
	wExtraBytesToRead := HTTP_UTF8.trailingBytesForUTF8[pbySource^];
	IF (pbySource + wExtraBytesToRead >= pbySourceEnd) THEN
		HTTP_UTF8toUTF16_3S := HTTP_UTF8.ERR_SOURCE_EXHAUSTED;
		EXIT;
	END_IF
	(* Do this check whether lenient or strict *)
	IF (NOT HTTP_IsLegalUTF8_3S(pbySource, WORD_TO_INT(wExtraBytesToRead+1)) AND xStrictConversion) THEN
		HTTP_UTF8toUTF16_3S := HTTP_UTF8.ERR_SOURCE_ILLEGAL;
		EXIT;
	END_IF
	(*
	* The cases all fall through. See "Note A" below.
	*)
	wExtraBytesToReadSave := wExtraBytesToRead;
	IF wExtraBytesToRead = 5 THEN
		dwSource := dwSource + pbySource^;
		pbySource := pbySource + 1;
		dwSource := SHL(dwSource, 6); (* remember, illegal UTF-8 *)
		wExtraBytesToRead := 4;
	END_IF
	IF wExtraBytesToRead = 4 THEN
		dwSource := dwSource + pbySource^;
		pbySource := pbySource + 1;
		dwSource := SHL(dwSource, 6); (* remember, illegal UTF-8 *)
		wExtraBytesToRead := 3;
	END_IF
	IF wExtraBytesToRead = 3 THEN
		dwSource := dwSource + pbySource^;
		pbySource := pbySource + 1;
		dwSource := SHL(dwSource, 6); 
		wExtraBytesToRead := 2;
	END_IF
	IF wExtraBytesToRead = 2 THEN
		dwSource := dwSource + pbySource^;
		pbySource := pbySource + 1;
		dwSource := SHL(dwSource, 6); 
		wExtraBytesToRead := 1;
	END_IF
	IF wExtraBytesToRead = 1 THEN
		dwSource := dwSource + pbySource^;
		pbySource := pbySource + 1;
		dwSource := SHL(dwSource, 6); 
		wExtraBytesToRead := 0;
	END_IF
	IF wExtraBytesToRead = 0 THEN
		dwSource := dwSource + pbySource^;
		pbySource := pbySource + 1;
	END_IF
	dwSource := dwSource - HTTP_UTF8.offsetsFromUTF8[wExtraBytesToReadSave];

	IF (pwTarget >= pwTargetEnd) THEN
		// We don't return the source yet: source -= (extraBytesToRead+1); /* Back up source POINTER! */
		HTTP_UTF8toUTF16_3S := HTTP_UTF8.ERR_TARGET_EXHAUSTED; 
		EXIT;
	END_IF
	IF (dwSource <= HTTP_UTF8.UNI_MAX_BMP) THEN 
		(* Target is a character <= 0xFFFF *)
		(* UTF-16 surrogate values are illegal in UTF-32 *)
		IF (dwSource >= HTTP_UTF8.UNI_SUR_HIGH_START AND dwSource <= HTTP_UTF8.UNI_SUR_LOW_END) THEN
			IF (xStrictConversion) THEN
				HTTP_UTF8toUTF16_3S := HTTP_UTF8.ERR_SOURCE_ILLEGAL;
				EXIT;
			ELSE 
				pwTarget^ := DWORD_TO_WORD(HTTP_UTF8.UNI_REPLACEMENT_CHAR);
				pwTarget := pwTarget + 2;
			END_IF
		ELSE
			pwTarget^ := DWORD_TO_WORD(dwSource); (* normal case *)
			pwTarget := pwTarget + 2;
		END_IF
	ELSIF (dwSource > HTTP_UTF8.UNI_MAX_UTF16) THEN
		IF (xStrictConversion) THEN
			HTTP_UTF8toUTF16_3S := HTTP_UTF8.ERR_SOURCE_ILLEGAL;
			// We don't return the source yet: source -= (extraBytesToRead+1); (* return to the start *)
			EXIT; (* Bail out; shouldn't continue *)
		ELSE 
			pwTarget^ := DWORD_TO_WORD(HTTP_UTF8.UNI_REPLACEMENT_CHAR);
			pwTarget := pwTarget + 2;
		END_IF
	ELSE 
		(* target is a character in range 0xFFFF - 0x10FFFF. *)
		IF (pwTarget + 1 >= pwTargetEnd) THEN
			// We don't return the source yet: source -= (extraBytesToRead+1); (* Back up source pointer! *)
			HTTP_UTF8toUTF16_3S := HTTP_UTF8.ERR_TARGET_EXHAUSTED; 
			EXIT;
		END_IF
		dwSource := dwSource - HTTP_UTF8.halfBase;
		pwTarget^ := DWORD_TO_WORD(SHR(dwSource, HTTP_UTF8.halfShift) + HTTP_UTF8.UNI_SUR_HIGH_START);
		pwTarget := pwTarget + 2;
		pwTarget^ := DWORD_TO_WORD(dwSource AND HTTP_UTF8.halfMask + HTTP_UTF8.UNI_SUR_LOW_START);
		pwTarget := pwTarget + 2;
	END_IF
END_WHILE

END_FUNCTION

// Functions/HTTP_IsLegalUTF8_3S
{attribute 'conditionalshow'}
FUNCTION HTTP_IsLegalUTF8_3S : BOOL
VAR_INPUT
 	pbySource 		: POINTER TO BYTE;
	iLength 		: INT;
END_VAR
VAR
	byX 			: BYTE;
	pbySourceEnd 	: POINTER TO BYTE;
END_VAR

HTTP_IsLegalUTF8_3S := FALSE;
pbySourceEnd := pbySource+TO_DWORD(iLength);
IF iLength = 4 OR iLength = 3 OR iLength = 2 OR iLength = 1 THEN
	IF iLength = 4 THEN
		pbySourceEnd := pbySourceEnd - 1;
		byX := pbySourceEnd^;
		IF (byX < 16#80 OR byX > 16#BF) THEN
			RETURN;
		END_IF
		iLength := 3;
	END_IF
	IF iLength = 3 THEN
		pbySourceEnd := pbySourceEnd - 1;
		byX := pbySourceEnd^;
		IF (byX < 16#80 OR byX > 16#BF) THEN
			RETURN;
		END_IF
		iLength := 2;
	END_IF
	IF iLength = 2 THEN
		pbySourceEnd := pbySourceEnd - 1;
		byX := pbySourceEnd^;
		IF (byX > 16#BF) THEN
			RETURN;
		END_IF
		
		CASE (pbySource^) OF
			(* no fbyXll-through in this inner switch *)
			16#E0: 
				IF (byX < 16#A0) THEN
					RETURN; 
				END_IF
			16#ED:  
				IF (byX > 16#9F) THEN
					RETURN; 
				END_IF
			16#F0:  
				IF (byX < 16#90) THEN
					RETURN; 
				END_IF
			16#F4:  
				IF (byX > 16#8F) THEN
					RETURN; 
				END_IF
		ELSE
			IF (byX < 16#80) THEN
				RETURN;
			END_IF
		END_CASE
		iLength := 1;
	END_IF
	IF iLength = 1 THEN
		IF (pbySource^ >= 16#80 AND pbySource^ < 16#C2) THEN
			RETURN;
		END_IF
	END_IF
ELSE
	RETURN;
END_IF
IF (pbySource^ > 16#F4) THEN
	RETURN;
END_IF
HTTP_IsLegalUTF8_3S := TRUE;

END_FUNCTION

// Functions/HTTP_Concat_3S
/// This function concatenates pchFrom to pstTo if the iBufferSize from pstTo is big enough. 
/// It will return FALSE and does no concatenation if one of the strings is NULL 
/// or the buffer size is not big enough.
{attribute 'conditionalshow'}
FUNCTION HTTP_Concat_3S : BOOL
VAR_INPUT
	pchFrom 		: CharBufferPtr;	// simply a pointer to byte
	pstTo 			: CharBufferPtr;		// simply a pointer to byte
	udiBufferSize 	: UDINT;			// the buffer size of pstTo
END_VAR
VAR
	{attribute 'ieccodeconversion_character_array'}
	pwFrom 			: POINTER TO WORD;
	{attribute 'ieccodeconversion_character_array'}
	pwTo 			: POINTER TO WORD;	
	diLengthFrom 	: DINT;
	diLengthTo 		: DINT;
	diForLoop		: DINT;
END_VAR

IF pchFrom = NULL OR pstTo = NULL THEN
	RETURN;		// return FALSE
END_IF

diLengthFrom := StrLenW(pchFrom);
diLengthTo := StrLenW(pstTo);

IF (diLengthTo * 2) + (diLengthFrom * 2) + 2 > UDINT_TO_DINT(udiBufferSize) THEN
	RETURN;		// return FALSE => result buffer not big enough
END_IF

pwFrom := pchFrom;
pwTo := pstTo;

// Concatenate the string pchFrom to pstTo
FOR diForLoop := 0 TO diLengthFrom - 1 DO
	pwTo[diLengthTo+diForLoop] := pwFrom[diForLoop];
END_FOR
// Set the string termination
pwTo[diLengthTo+diForLoop] := 0;
HTTP_Concat_3S := TRUE;

END_FUNCTION

// ChangeLog
PROGRAM ChangeLog
VAR
END_VAR

{attribute 'conditionalshow'}
//Library based on 3S - Smart Software Solutions HTTP Client, available from:
//https://store.codesys.com/http-client-example.html
//All credits go to 3S and their library.

//V1.2.200929
//Removed unused variables and added pragma to satisfy static analysis on used variables.

//V1.2 - April 2020:
//Removed error parsing of StringToURL.
//Cleaned eError list (unused functions).
//Compiler update to 3.5.14.40.
//Added TCP handler errors (with corresponding offset to match library).

//V1.1 - Feb 2019:
//Changed some constants into properties.
//Added conditionalshow attribute.
//Added result valid to compare size in header and actual size.

//V1.0 - Dec 2018:
//Library provides an easier interface for the function block in the 3S library.

END_PROGRAM
